TYPE DUT_EL1918_Logic :
STRUCT
	
	inbyte_1			:BYTE;
	inbyte_2			:BYTE;
	outbyte_1			:BYTE;

	       
END_STRUCT
END_TYPE

(* stored: Version 1.1.0.1
   DUT DUT_EL1918_Logic: Id {05bc814b-fd37-4087-b46f-5757f8ea4031} *)
